Universal Robots PolyScope program: ANGEL.urp

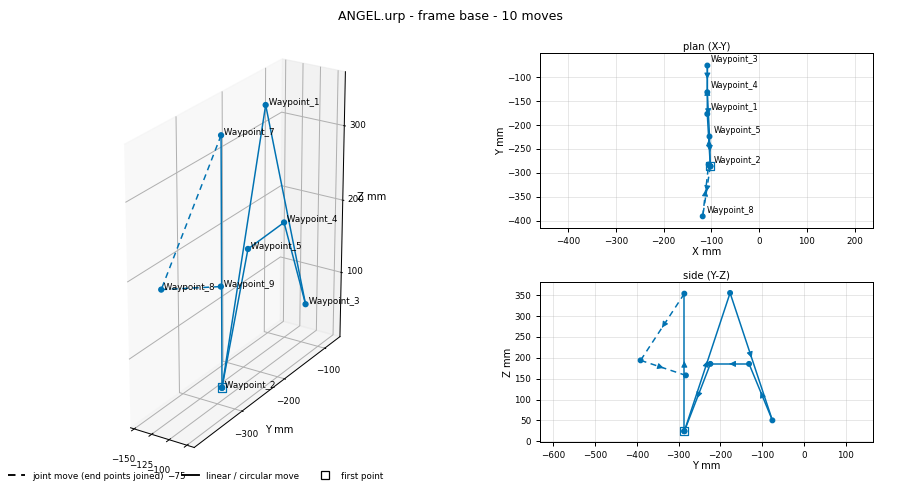
[picture p0: tool path of ANGEL.urp in frame base, 10 of 10 moves have a stored position in this frame; points joined in program order, loops and branches not executed]
Program ANGEL (installation=default directory=/ursim/programs createdIn=3.15.8.106339 lastSavedIn=3.15.8.106339 robotSerialNumber=2018359999)
Calibrated DH parameters: a=[0, -0.425, -0.39225, 0, 0, 0]; d=[0.089159, 0, 0, 0.10915, 0.09465, 0.0823]; alpha=[1.570796, 0, 0, 1.570796, -1.570796, 0]; deltaTheta=[0, 0, 0, 0, 0, 0]
Robot Program (runOnlyOnce=false)
  Popup Message (haltProgram=false message=Se dibujara la letra A y P inputType=Text)
  MoveL speed 250 mm/s, acceleration 1200 mm/s^2 (useActiveTCP=true) feature=Base
    Waypoint Waypoint_2: TCP in base x=-102.039 y=-286.26 z=24.122 mm, rx=0.0207 ry=-3.0547 rz=-0.6611 rad; joints [-88.448, -102.315, -146.678, -45.442, 89.579, 0.866] deg
    Waypoint Waypoint_1: TCP in base x=-108.371 y=-176.691 z=355.227 mm, rx=-0.0149 ry=2.7127 rz=-1.5687 rad; joints [-90.098, -38.671, -147.252, -24, 90.754, -0.293] deg
    Waypoint Waypoint_3: TCP in base x=-108.197 y=-75.347 z=50.03 mm, rx=-0.0093 ry=3.066 rz=-0.6301 rad; joints [-90.098, -38.671, -184.105, -24, 90.754, -0.293] deg
    Waypoint Waypoint_4: TCP in base x=-108.293 y=-131.249 z=185.335 mm, rx=-0.0128 ry=2.8895 rz=-1.2085 rad; joints [-90.098, -31.912, -168.698, -24, 90.754, -0.293] deg
    Waypoint Waypoint_5: TCP in base x=-103.729 y=-223.898 z=185.335 mm, rx=-0.0128 ry=2.8895 rz=-1.2085 rad; joints [-88.448, -71.246, -162.387, 9.025, 89.579, 0.866] deg
    Waypoint Waypoint_2: TCP in base x=-102.039 y=-286.26 z=24.122 mm, rx=0.0207 ry=-3.0547 rz=-0.6611 rad; joints [-88.448, -102.315, -146.678, -45.442, 89.579, 0.866] deg
    Waypoint Waypoint_6: TCP in base x=-102.039 y=-286.26 z=24.122 mm, rx=0.0207 ry=-3.0547 rz=-0.6611 rad; joints [-88.448, -102.315, -146.678, -45.442, 89.579, 0.866] deg
    Waypoint Waypoint_7: TCP in base x=-102.039 y=-286.26 z=353.557 mm, rx=0.0207 ry=-3.0547 rz=-0.6611 rad; joints [-88.448, -67.782, -114.404, -112.248, 89.579, 0.866] deg
    MoveJ speed 60 deg/s, acceleration 80 deg/s^2 (useActiveTCP=true)
      Waypoint Waypoint_8: TCP in base x=-117.986 y=-391.004 z=193.789 mm, rx=0.0217 ry=-2.4546 rz=-1.9094 rad; joints [-90.738, -104.75, -104.959, -136.05, 87.359, 0.303] deg
      Waypoint Waypoint_9: TCP in base x=-105.543 y=-282.522 z=157.793 mm, rx=0.0217 ry=-2.4546 rz=-1.9094 rad; joints [-88.99, -93.98, -124.369, -127.424, 89.054, 0.733] deg
